TYPE ST160_Recipe_t :
STRUCT
    Use_left_160 : BOOL; //a 
    Use_right_160 : BOOL; // 
    Use_left_165 : BOOL; // b
    Use_right_165 : BOOL; // 
END_STRUCT
END_TYPE

(* stored: Version 1.1.0.1, ProductVersion 3.1.4024.6
   DUT ST160_Recipe_t: Id {34ae7bc1-90d5-4547-bc33-0df5746ede05} *)
